{attribute 'GeneratedUsingTerminal: EL3413-0000-0019'}
{attribute addProperty BoxType "EL3413-0000-0019"}
{attribute addProperty Id "STATUSAT %I*STATUS_58431BA93IndexAT %I*USINT1ChannelAT %I*USINT1ValueAT %I*DINT4"}
{attribute addProperty CRC "912382829"}
{attribute addProperty Size "9"}
TYPE PM_Inputs_Auxiliary_3661DB6D EXTENDS InputBase_8311D824 :
STRUCT
	{attribute addProperty Name "STATUS"}
	STATUS AT %I* : STATUS_58431BA9;
	{attribute addProperty Name "Index"}
	Index AT %I* : USINT;
	{attribute addProperty Name "Channel"}
	Channel AT %I* : USINT;
	{attribute addProperty Name "Value"}
	Value AT %I* : DINT;
END_STRUCT
END_TYPE

(* stored: Version 1.2.0.0, ProductVersion 3.1.4024.11
   DUT PM_Inputs_Auxiliary_3661DB6D: Id {4ca66b79-e35b-4868-a57a-c060b785940a} *)
